(* CoDeSys 2.3.10.0 project: TwinCAT NC Sample Superposition.pro *)
(* Libraries: STANDARD.LIB 5.6.98 12:03:02, TcBase.lib*14.5.09 12:14:08, TcSystem.lib*18.2.11 17:15:48, TcBaseMath.lib 27.7.04 12:07:56, TcMath.lib 23.9.04 15:15:30, TcMC2.lib*28.3.11 08:59:11 *)

(* Task configuration *)
TASK Standard (PRIORITY := 0, INTERVAL := T#10ms);
	MAIN
END_TASK

(* Global variable list: TwinCAT_Configuration *)
(* Generated automatically by TwinCAT - (read only) *)
VAR_CONFIG
	MAIN.Axis1.PlcToNc AT %QB0 : PLCTONC_AXIS_REF;
	MAIN.Axis1.NcToPlc AT %IB0 : NCTOPLC_AXIS_REF;	(*  ~ {LinkedWith:TINC^NC-Task 1 SAF^Axes^Axis 1^Outputs^Axis 1_ToPlc} *)
	MAIN.Axis2.PlcToNc AT %QB128 : PLCTONC_AXIS_REF;
	MAIN.Axis2.NcToPlc AT %IB128 : NCTOPLC_AXIS_REF;
END_VAR

(* Data type *)
TYPE MoveState_t :
(
	MOVESTATE_INIT,
	MOVESTATE_ENABLE,
	MOVESTATE_COUPLE,
	MOVESTATE_DECOUPLE,
	MOVESTATE_FORWARD,
	MOVESTATE_SUPERPOSITION,
	MOVESTATE_BACKWARDS,
	MOVESTATE_ERROR,
	MOVESTATE_RESET
);
END_TYPE

(* POU MAIN, ST *)
PROGRAM MAIN
VAR
	Axis1 : AXIS_REF;					(* axis reference data structure *)
	Axis2 : AXIS_REF;					(* axis reference data structure *)

	state: MoveState_t;				(* state machine state *)

	PowerAxis1: MC_Power;
	PowerAxis1Out: ST_McOutputs;		(* debug function block output data *)

	MoveAbsolute1: MC_MoveAbsolute;
	MoveAbsolute1Out: ST_McOutputs;	(* debug function block output data *)
	MoveAbsolute2: MC_MoveAbsolute;
	MoveAbsolute2Out: ST_McOutputs;	(* debug function block output data *)

	Reset1: MC_Reset;
	Reset1Out : ST_McOutputs;			(* debug function block output data *)
	Reset2: MC_Reset;
	Reset2Out : ST_McOutputs;			(* debug function block output data *)

	PowerAxis2: MC_Power;
	PowerAxis2Out: ST_McOutputs;
	GearIn: MC_GearIn;
	GearInOut: ST_McOutputs;
	MoveSuperImposed: MC_MoveSuperImposed;
	MoveSuperImposedOut: ST_McOutputs;
	GearOut: MC_GearOut;
	GearOutOut: ST_McOutputs;

	(* output data *)
	MoveSuperImposed_Warning: BOOL;
	MoveSuperImposed_WarningID: UDINT;
	MoveSuperImposed_ActualVelocityDiff: LREAL;
	MoveSuperImposed_ActualDistance: LREAL;
	MoveSuperImposed_ActualLength: LREAL;
	MoveSuperImposed_ActualAcceleration: LREAL;
	MoveSuperImposed_ActualDeceleration: LREAL;
END_VAR
	(* update the axis status at the beginning of each cycle *)
	Axis1.ReadStatus;
	Axis2.ReadStatus;

	(* move axis using a state machine *)
	CASE state OF

		MOVESTATE_INIT :	(* initialisation *)
			(* initialize all function blocks *)
			MoveAbsolute1.Execute := FALSE;
			MoveAbsolute2.Execute := FALSE;
			Reset1.Execute := FALSE;
			Reset2.Execute := FALSE;
			GearIn.Execute := FALSE;
			GearOut.Execute := FALSE;
			MoveSuperimposed.Execute := FALSE;
			state := MOVESTATE_ENABLE;

		MOVESTATE_ENABLE :
			PowerAxis1.Enable := TRUE;
			PowerAxis1.Enable_Positive := TRUE;
			PowerAxis1.Enable_Negative := TRUE;
			PowerAxis2.Enable := TRUE;
			PowerAxis2.Enable_Positive := TRUE;
			PowerAxis2.Enable_Negative := TRUE;
			IF PowerAxis1.Status AND PowerAxis2.Status THEN
				state := MOVESTATE_COUPLE;
			ELSIF PowerAxis1.Error OR PowerAxis2.Error THEN
				state := MOVESTATE_ERROR;
			END_IF

		MOVESTATE_COUPLE :
			GearIn.Execute := TRUE;
			IF GearIn.InGear THEN
				state := MOVESTATE_FORWARD;
			END_IF

		MOVESTATE_FORWARD :		(* start to first position *)
			MoveAbsolute1.Position := 1500;		(* start to intermediate tartet position *)
			MoveAbsolute1.Velocity := 500;		(* medium velocity level *)
			MoveAbsolute1.BufferMode := MC_Buffered;
			MoveAbsolute1.Execute := TRUE;
			IF MoveAbsolute1.Active  THEN
				(* axis is executing job but is not yet finished *)
				MoveAbsolute1.Execute := FALSE;
				(* leave this state and buffer a second command *)
				state := MOVESTATE_SUPERPOSITION;
			ELSIF MoveAbsolute1.CommandAborted OR MoveAbsolute1.Error THEN
				state := MOVESTATE_ERROR;
			END_IF

		MOVESTATE_SUPERPOSITION :
			IF Axis1.NcToPlc.SetPos > 500 THEN
				MoveSuperimposed.Distance := 100;
				MoveSuperimposed.Length := 500;
				MoveSuperimposed.Mode := SUPERPOSITIONMODE_VELOREDUCTION_ADDITIVEMOTION;
				MoveSuperimposed.VelocityDiff := 500;
				MoveSuperimposed.VelocityProcess := Axis2.NcToPlc.SetVelo;
				MoveSuperimposed.Execute := TRUE;
			END_IF
			IF MoveSuperimposed.Done AND MoveAbsolute1.Done THEN
				state := MOVESTATE_DECOUPLE;
			END_IF

		MOVESTATE_DECOUPLE :
			GearOut.Execute := TRUE;
			IF GearOut.Done THEN
				state := MOVESTATE_BACKWARDS;
			END_IF

		MOVESTATE_BACKWARDS :	(* move back to initial position *)
			MoveAbsolute1.Position := 0;		(* position close to initial position *)
			MoveAbsolute1.Velocity := 2000;		(* high velocity *)
			MoveAbsolute1.Execute := TRUE;
			MoveAbsolute2.Position := 0;		(* position close to initial position *)
			MoveAbsolute2.Velocity := 2000;		(* high velocity *)
			MoveAbsolute2.Execute := TRUE;
			IF MoveAbsolute1.Done AND MoveAbsolute2.Done THEN
				(* axis is executing job but is not yet finished *)
				MoveAbsolute1.Execute := FALSE;
				(* leave this state and buffer a second command *)
				state := MOVESTATE_INIT;
			ELSIF MoveAbsolute1.CommandAborted OR MoveAbsolute1.Error
				OR  MoveAbsolute2.CommandAborted OR MoveAbsolute2.Error
				THEN
				state := MOVESTATE_ERROR;
			END_IF

		MOVESTATE_ERROR :
			IF Axis1.Status.Error OR Axis2.Status.Error THEN
				state := MOVESTATE_RESET;	(* axis error requires reset *)
			ELSE
				state := MOVESTATE_INIT;		(* function block errors don't need a reset *)
			END_IF

		MOVESTATE_RESET :
			Reset1.Execute := TRUE;
			Reset2.Execute := TRUE;
			IF Reset1.Done AND Reset2.Done THEN
				state := MOVESTATE_INIT;
			ELSIF Reset1.Error OR Reset2.Error THEN
				state := MOVESTATE_INIT; (* can't do anything here *)
			END_IF

	END_CASE

	ActPower;		(* call the power function block *)
	ActMove;		(* call the move function block *)
	ActReset;		(* call the reset function block *)
	ActCouple;		(* call the master slave coupling function block *)
	ActSuperposition;	(* call the superposition function block *)
END_PROGRAM
ACTION ActCouple:
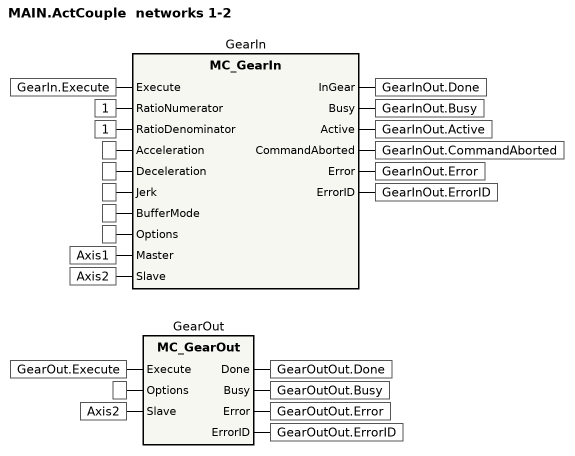
_FBD_ (* Function Block Diagram *)
NETWORK 1
	GearIn:MC_GearIn(Execute: GearIn.Execute, RatioNumerator: 1, RatioDenominator: 1, Acceleration: , Deceleration: , Jerk: , BufferMode: , Options: , Master: Axis1, Slave: Axis2, Busy => GearInOut.Busy, Active => GearInOut.Active, CommandAborted => GearInOut.CommandAborted, Error => GearInOut.Error, ErrorID => GearInOut.ErrorID) => GearInOut.Done
NETWORK 2
	GearOut:MC_GearOut(Execute: GearOut.Execute, Options: , Slave: Axis2, Busy => GearOutOut.Busy, Error => GearOutOut.Error, ErrorID => GearOutOut.ErrorID) => GearOutOut.Done
_END_FBD_
END_ACTION
ACTION ActMove:
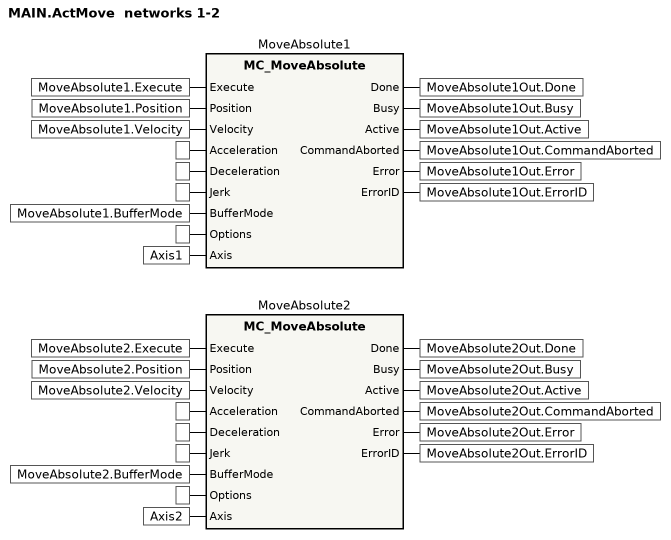
_FBD_ (* Function Block Diagram *)
NETWORK 1
	MoveAbsolute1:MC_MoveAbsolute(Execute: MoveAbsolute1.Execute, Position: MoveAbsolute1.Position, Velocity: MoveAbsolute1.Velocity, Acceleration: , Deceleration: , Jerk: , BufferMode: MoveAbsolute1.BufferMode, Options: , Axis: Axis1, Busy => MoveAbsolute1Out.Busy, Active => MoveAbsolute1Out.Active, CommandAborted => MoveAbsolute1Out.CommandAborted, Error => MoveAbsolute1Out.Error, ErrorID => MoveAbsolute1Out.ErrorID) => MoveAbsolute1Out.Done
NETWORK 2
	MoveAbsolute2:MC_MoveAbsolute(Execute: MoveAbsolute2.Execute, Position: MoveAbsolute2.Position, Velocity: MoveAbsolute2.Velocity, Acceleration: , Deceleration: , Jerk: , BufferMode: MoveAbsolute2.BufferMode, Options: , Axis: Axis2, Busy => MoveAbsolute2Out.Busy, Active => MoveAbsolute2Out.Active, CommandAborted => MoveAbsolute2Out.CommandAborted, Error => MoveAbsolute2Out.Error, ErrorID => MoveAbsolute2Out.ErrorID) => MoveAbsolute2Out.Done
_END_FBD_
END_ACTION
ACTION ActPower:
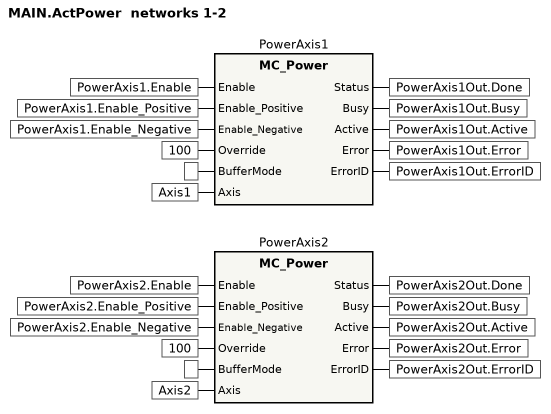
_FBD_ (* Function Block Diagram *)
NETWORK 1
	PowerAxis1:MC_Power(Enable: PowerAxis1.Enable, Enable_Positive: PowerAxis1.Enable_Positive, Enable_Negative: PowerAxis1.Enable_Negative, Override: 100, BufferMode: , Axis: Axis1, Busy => PowerAxis1Out.Busy, Active => PowerAxis1Out.Active, Error => PowerAxis1Out.Error, ErrorID => PowerAxis1Out.ErrorID) => PowerAxis1Out.Done
NETWORK 2
	PowerAxis2:MC_Power(Enable: PowerAxis2.Enable, Enable_Positive: PowerAxis2.Enable_Positive, Enable_Negative: PowerAxis2.Enable_Negative, Override: 100, BufferMode: , Axis: Axis2, Busy => PowerAxis2Out.Busy, Active => PowerAxis2Out.Active, Error => PowerAxis2Out.Error, ErrorID => PowerAxis2Out.ErrorID) => PowerAxis2Out.Done
_END_FBD_
END_ACTION
ACTION ActReset:
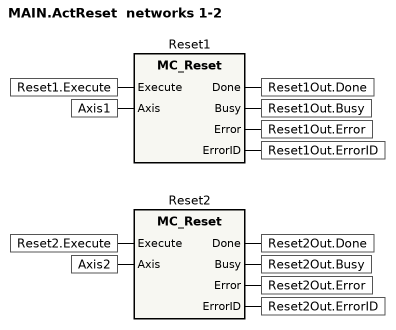
_FBD_ (* Function Block Diagram *)
NETWORK 1
	Reset1:MC_Reset(Execute: Reset1.Execute, Axis: Axis1, Busy => Reset1Out.Busy, Error => Reset1Out.Error, ErrorID => Reset1Out.ErrorID) => Reset1Out.Done
NETWORK 2
	Reset2:MC_Reset(Execute: Reset2.Execute, Axis: Axis2, Busy => Reset2Out.Busy, Error => Reset2Out.Error, ErrorID => Reset2Out.ErrorID) => Reset2Out.Done
_END_FBD_
(* the same logic as Structured Text *)
(* Network 1 *)
Reset1(Execute := Reset1.Execute, Axis := Axis1);
Reset1Out.Busy := Reset1.Busy;
Reset1Out.Error := Reset1.Error;
Reset1Out.ErrorID := Reset1.ErrorID;
Reset1Out.Done := Reset1.Done;
(* Network 2 *)
Reset2(Execute := Reset2.Execute, Axis := Axis2);
Reset2Out.Busy := Reset2.Busy;
Reset2Out.Error := Reset2.Error;
Reset2Out.ErrorID := Reset2.ErrorID;
Reset2Out.Done := Reset2.Done;
END_ACTION
ACTION ActSuperposition:
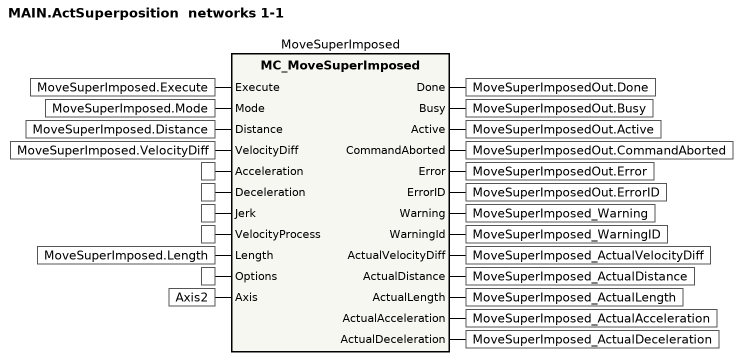
_FBD_ (* Function Block Diagram *)
NETWORK 1
	MoveSuperImposed:MC_MoveSuperImposed(Execute: MoveSuperImposed.Execute, Mode: MoveSuperImposed.Mode, Distance: MoveSuperImposed.Distance, VelocityDiff: MoveSuperImposed.VelocityDiff, Acceleration: , Deceleration: , Jerk: , VelocityProcess: , Length: MoveSuperImposed.Length, Options: , Axis: Axis2, Busy => MoveSuperImposedOut.Busy, Active => MoveSuperImposedOut.Active, CommandAborted => MoveSuperImposedOut.CommandAborted, Error => MoveSuperImposedOut.Error, ErrorID => MoveSuperImposedOut.ErrorID, Warning => MoveSuperImposed_Warning, WarningId => MoveSuperImposed_WarningID, ActualVelocityDiff => MoveSuperImposed_ActualVelocityDiff, ActualDistance => MoveSuperImposed_ActualDistance, ActualLength => MoveSuperImposed_ActualLength, ActualAcceleration => MoveSuperImposed_ActualAcceleration, ActualDeceleration => MoveSuperImposed_ActualDeceleration) => MoveSuperImposedOut.Done
_END_FBD_
END_ACTION
